{attribute 'TcGenerated'}
{attribute 'no-analysis'}
{attribute 'linkalways'}
// This function has been automatically generated from the project information.
VAR_GLOBAL CONSTANT
	{attribute 'const_non_replaced'}
	stLibVersion_HomePLC_Logging : ST_LibVersion := (iMajor := 1, iMinor := 0, iBuild := 1, iRevision := 0, nFlags := 0, sVersion := '1.0.1');
END_VAR

(* stored: Version 1.1.0.1, ProductVersion 3.1.4024.12
   GVL Global_Version: Id {8856f283-1fcf-44d5-a835-a739fc0d16f2} *)
